(* IEC 61131-3 sources: RIA_practicals/openplc/build, 2 files *)

(* ---- plc.st ---- *)
TYPE
  LOGLEVEL : (CRITICAL, WARNING, INFO, DEBUG) := INFO;
END_TYPE

FUNCTION_BLOCK LOGGER
  VAR_INPUT
    TRIG : BOOL;
    MSG : STRING;
    LEVEL : LOGLEVEL := INFO;
  END_VAR
  VAR
    TRIG0 : BOOL;
  END_VAR

  IF TRIG AND NOT TRIG0 THEN
  {{
   LogMessage(GetFbVar(LEVEL),(char*)GetFbVar(MSG, .body),GetFbVar(MSG, .len));
  }}
  END_IF;
  TRIG0:=TRIG;
END_FUNCTION_BLOCK

PROGRAM blinky_psy
  VAR
    blinky_led AT %QX0.3 : BOOL;
  END_VAR
  VAR
    TON0 : TON;
    TOF0 : TOF;
  END_VAR

  TON0(EN := TRUE, IN := NOT(blinky_led), PT := T#500ms);
  TOF0(EN := TON0.ENO, IN := TON0.Q, PT := T#500ms);
  blinky_led := TOF0.Q;
END_PROGRAM

CONFIGURATION Config0

  RESOURCE Res0 ON PLC
    TASK task0(INTERVAL := T#20ms,PRIORITY := 0);
    PROGRAM instance0 WITH task0 : blinky_psy;
  END_RESOURCE
END_CONFIGURATION

(* ---- generated_plc.st ---- *)
PROGRAM blinky_psy
  VAR
    blinky_led AT %QX0.3 : BOOL;
  END_VAR
  VAR
    TON0 : TON;
    TOF0 : TOF;
  END_VAR

  TON0(EN := TRUE, IN := NOT(blinky_led), PT := T#500ms);
  TOF0(EN := TON0.ENO, IN := TON0.Q, PT := T#500ms);
  blinky_led := TOF0.Q;
END_PROGRAM

CONFIGURATION Config0

  RESOURCE Res0 ON PLC
    TASK task0(INTERVAL := T#20ms,PRIORITY := 0);
    PROGRAM instance0 WITH task0 : blinky_psy;
  END_RESOURCE
END_CONFIGURATION
